FUNCTION_BLOCK UT_AuxiliaryInputMapping_Type_14_BidirectionalCounter (* Type 14 BidirectionalCounter Count increases when turning in the encoders &quot;increase&quot; direction (analog opposite direction) *)
  (* Standard: ISO 11783-6; Classification: AUX – ISO 11783-6; Function: All Inputs; Type: UT according to ISO 11783-6; Description: Copyright (c) 2018, 2023 Jose Cabral, HR Agrartechnik GmbH This program and the accompanying materials are made available under the terms of the Eclipse Public License 2.0 which is available at https://www.eclipse.org/legal/epl-2.0/ SPDX-License-Identifier: EPL-2.0 - Type 14 BidirectionalCounter Count increases when turning in the encoders "increase" direction (analog opposite direction) Applicable AUX-N only * maps to IW IW - Input WORD (16 Bit) *)
  (* Version 1.0, 2018-12-05, Jose Cabral *)
  (* Version 1.1, 2022-08-04, Franz Höpfinger, HR Agrartechnik GmbH *)
  (* Version 1.2, 2023-01-05, Franz Höpfinger, HR Agrartechnik GmbH *)
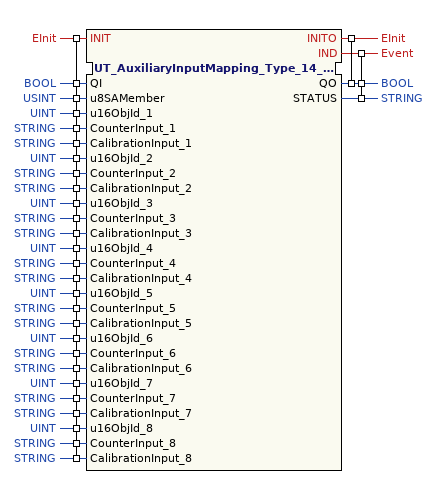
  EVENT_INPUT
    INIT : EInit WITH QI, u8SAMember, u16ObjId_1, CounterInput_1, CalibrationInput_1, u16ObjId_2, CounterInput_2, CalibrationInput_2, u16ObjId_3, CounterInput_3, CalibrationInput_3, u16ObjId_4, CounterInput_4, CalibrationInput_4, u16ObjId_5, CounterInput_5, CalibrationInput_5, u16ObjId_6, CounterInput_6, CalibrationInput_6, u16ObjId_7, CounterInput_7, CalibrationInput_7, u16ObjId_8, CounterInput_8, CalibrationInput_8; (* Service Initialization *)
  END_EVENT
  EVENT_OUTPUT
    INITO : EInit WITH QO; (* Initialization Confirm *)
    IND WITH QO, STATUS; (* Indication from Resource *)
  END_EVENT
  VAR_INPUT
    QI : BOOL; (* Event Input Qualifier *)
    u8SAMember : USINT := GLOBAL; (* Dummy !, set to GLOBAL if in doubt. OFF deactivates FB. *)
    u16ObjId_1 : UINT; (* Object ID of Input 1 *)
    CounterInput_1 : STRING; (* Identifier for Input 1 Current Count *)
    CalibrationInput_1 : STRING; (* Calibration — Encoder Counts per revolution *)
    u16ObjId_2 : UINT; (* Object ID of Input 2 *)
    CounterInput_2 : STRING; (* Identifier for Input 2 Current Count *)
    CalibrationInput_2 : STRING; (* Calibration — Encoder Counts per revolution *)
    u16ObjId_3 : UINT; (* Object ID of Input 3 *)
    CounterInput_3 : STRING; (* Identifier for Input 3 Current Count *)
    CalibrationInput_3 : STRING; (* Calibration — Encoder Counts per revolution *)
    u16ObjId_4 : UINT; (* Object ID of Input 4 *)
    CounterInput_4 : STRING; (* Identifier for Input 4 Current Count *)
    CalibrationInput_4 : STRING; (* Calibration — Encoder Counts per revolution *)
    u16ObjId_5 : UINT; (* Object ID of Input 5 *)
    CounterInput_5 : STRING; (* Identifier for Input 5 Current Count *)
    CalibrationInput_5 : STRING; (* Calibration — Encoder Counts per revolution *)
    u16ObjId_6 : UINT; (* Object ID of Input 6 *)
    CounterInput_6 : STRING; (* Identifier for Input 6 Current Count *)
    CalibrationInput_6 : STRING; (* Calibration — Encoder Counts per revolution *)
    u16ObjId_7 : UINT; (* Object ID of Input 7 *)
    CounterInput_7 : STRING; (* Identifier for Input 7 Current Count *)
    CalibrationInput_7 : STRING; (* Calibration — Encoder Counts per revolution *)
    u16ObjId_8 : UINT; (* Object ID of Input 8 *)
    CounterInput_8 : STRING; (* Identifier for Input 8 Current Count *)
    CalibrationInput_8 : STRING; (* Calibration — Encoder Counts per revolution *)
  END_VAR
  VAR_OUTPUT
    QO : BOOL; (* Event Output Qualifier *)
    STATUS : STRING; (* Service Status *)
  END_VAR
END_FUNCTION_BLOCK
